// TwinCAT 3 PLC project VisionPLC
// ProgramVersion: 3.1.4024.0
// libraries:
//   Tc2_Standard, * (Beckhoff Automation GmbH)
//   Tc2_System, * (Beckhoff Automation GmbH)
//   Tc2_Utilities, * (Beckhoff Automation GmbH)
//   Tc3_Module, * (Beckhoff Automation GmbH)
//   Tc3_Vision, * (Beckhoff Automation GmbH)
// project tree:
//   DUTs/ ST_CSV_Record.TcDUT
//   GVLs/ GVL.TcGVL
//   / PlcTask.TcTTO
//   POUs/ Barcode.TcPOU, MAIN.TcPOU, P_TextModeWrite.TcPOU, QRCODE.TcPOU
// real-time tasks:
//   TASK PlcTask: cycle T#10ms, priority 20, ADS port 350
//   TASK VnTask ImgAcq (FileSource1): cycle T#10ms, priority 5, ADS port 351

CONFIGURATION VisionPLC
    RESOURCE PLC ON TwinCAT3
        TASK PlcTask(INTERVAL := T#10ms, PRIORITY := 20);
        PROGRAM MAIN WITH PlcTask : MAIN;
    END_RESOURCE
END_CONFIGURATION

// ---- DUTs/ST_CSV_Record.TcDUT
TYPE ST_CSV_Record :
STRUCT
sName 	: T_MaxString 	:= '';
	nNumber	: UDINT 		:= 0;
	fPos	: LREAL 		:= 0.0;
	bOP		: BOOL 			:= FALSE;
	sDesc	: STRING(40)	:= '';
	data	: ARRAY[0..7] OF BYTE;
END_STRUCT
END_TYPE

// ---- GVLs/GVL.TcGVL
{attribute 'qualified_only'}
VAR_GLOBAL CONSTANT
	MAX_CSV_ROWS 			: UDINT := 10;
	MAX_CSV_COLUMNS 		: UDINT := 5;
	MAX_CSV_FIELD_LENGTH	: UDINT := 100;
END_VAR

// ---- POUs/MAIN.TcPOU

PROGRAM MAIN
VAR
	//fbfilesource                                    : FB_VN_FileSourceControl;	
	CAMERA 											: FB_VN_FileSourceControl;	
	raw_image										: ITcVnImage;	
	WORKED_image										: ITcVnImage;	
	ipImageIn              						    :   ITcVnImage;
	display_raw_image								: ITcVnDisplayableImage;		
	
	ipcontours										: ITcVnContainer;	
	number_of_elements								: ULINT;	
	hr, hr1											: HRESULT;	
	cState 											: ETcVnCameraState;	
	green_color										: TcVnVector4_LREAL := [0,255,0,0];	
	Bcolor										: TcVnVector4_LREAL := [100,0,0,0];
	stext											: STRING;
	
	
//	raw_image           :    ITcVnImage;

// QR Code
ipCodeDecodedList   :    ITcVnContainer; 
ipCodeContourList   :    ITcVnContainer;
sCodeAsString       :    STRING(255);


// Output
//sText               :    STRING;

// Color
aColorRed           :    TcVnVector4_LREAL := [255, 0, 0];
pCodeDecodedList         :   ITcVnContainer; 


eBarcodeSearchDirection   :   ETcVnBarcodeSearchDirection := TCVN_BSD_ANY;
eBarcodeType              :   ETcVnBarcodeType := TCVN_BT_EAN13;
display_barcode								: ITcVnDisplayableImage;
ipImageRes: ITcVnImage;	




// Color
aColorgreen                 :   TcVnVector4_LREAL := [0, 255, 0];

//pwrite variable
bChangeSeparatorToComma	: BOOL := FALSE;
END_VAR

IF bChangeSeparatorToComma THEN
	DEFAULT_CSV_FIELD_SEP := 16#2C;(* Comma ASCII code *)
ELSE
	DEFAULT_CSV_FIELD_SEP := 16#3B;(* Semicolon ASCII code *)
END_IF




//camera code 
cState 				:= CAMERA.GetState();

CASE cState OF
	

TCVN_CS_INITIAL, TCVN_CS_OPENING, TCVN_CS_OPENED, TCVN_CS_STARTACQUISITION :

 	hr  := CAMERA.StartAcquisition();  // start Camera acquisition



TCVN_CS_ACQUIRING:
	HR := CAMERA.GetCurrentImage(raw_image);   //get image from file source 
	ipImageIn := raw_image;   //get image from file source 
	
	 IF SUCCEEDED(HR) AND ipImageIn <> 0 THEN
		 
		
// Check if the function was executed successfully 	

		

		(*hr := F_VN_ConvertColorSpace(raw_image, worked_image, TCVN_CST_RGB_TO_GRAY, hr);
		hr := F_VN_FindContours(worked_image, ipcontours, hr);
		hr := F_VN_GetNumberOfElements(ipcontours,number_of_elements, hr);
		hr := F_VN_DrawContours(ipcontours,-1,raw_image,green_color,2, hr);
		
		stext := ULINT_TO_STRING(number_of_elements);
		
		hr := F_VN_PutText(STEXT, raw_image, 70,270,TCVN_FT_HERSHEY_COMPLEX,2 , Bcolor, hr);
		
	END_IF

		hr :=  F_VN_CopyIntoDisplayableImage(raw_image, display_raw_image, hr); *)
	
 		
	//Barcode();	
 	QRCODE();
	 	END_IF

TCVN_CS_ERROR:	

	hr 	:= CAMERA.Reset();
END_CASE

END_PROGRAM

// ---- POUs/QRCODE.TcPOU
PROGRAM QRCODE
VAR
	hr              :    HRESULT;
	hr1				: HRESULT;
raw_image           :    ITcVnImage;
ipImageInDisp       :    ITcVnDisplayableImage;

ipImageResQR        :    ITcVnImage;
ipImageResDisp      :    ITcVnDisplayableImage;


// QR Code
ipCodeDecodedList   :    ITcVnContainer; 
ipCodeContourList   :    ITcVnContainer;
sCodeAsString       :    STRING(255);

// Watchdog
hrWD                :    HRESULT;
tStop               :    DINT := 20000;
tRest               :    DINT;

// Output
sText               :    STRING;

// Color
aColorRed           :    TcVnVector4_LREAL := [255, 0, 0];
aColorblue          :    TcVnVector4_LREAL := [0, 0, 255];

//string array
database1			: ARRAY[0..GVL.MAX_CSV_ROWS] OF STRING(GVL.MAX_CSV_FIELD_LENGTH);
i					: INT:=0 ;
j					: INT := 0;


	v1: STRING;
END_VAR

ipImageResQR := main.raw_image;
hr := F_VN_ReadQRCodeExp(main.raw_image, ipCodeDecodedList, ipCodeContourList, 1, TCVN_CSS_ONLY_NOT_INVERTED + TCVN_CSS_ONLY_NOT_FLIPPED, main.hr);
// Check if the function was executed successfully 
IF hr = S_OK THEN
    // Export Code into String
	hr 			:= F_VN_ExportSubContainer_String(ipCodeDecodedList, 0, sCodeAsString, 255, hr);
	P_TextModeWrite();
	

    // Write Code into Result Image
    hr := F_VN_PutTextExp(sCodeAsString,main.raw_image, 50, 50, ETcVnFontType.TCVN_FT_HERSHEY_PLAIN, 1, aColorRed,3, TCVN_LT_4_CONNECTED, FALSE, hr);

    // Draw Code Contour into Result Image
	 hr := F_VN_DrawContours(ipCodeContourList, -1, main.raw_image, aColorRed, 3, main.hr); 

    // Write HRESULT into Result Image
    sText := ('Qrcode read '); 
	hr := F_VN_PutTextExp(sText, main.raw_image, 200,240, ETcVnFontType.TCVN_FT_HERSHEY_PLAIN, 1, aColorblue,3, TCVN_LT_4_CONNECTED, FALSE, hr);
	hr :=  F_VN_CopyIntoDisplayableImage(main.raw_image, main.display_raw_image,hr);
	

	//hr1 := F_VN_PutTextExp(sText, ipImageRes, 60,240, ETcVnFontType.TCVN_FT_HERSHEY_PLAIN, 1, aColorblue,3, TCVN_LT_4_CONNECTED, FALSE, hr1);
	hr :=  F_VN_CopyIntoDisplayableImage(ipImageResQR, ipImageResDisp,hr);
ELSE
    // Write HRESULT into Result Image
    sText := CONCAT('QR cannot be read ', DINT_TO_STRING(hr)); 
    hr := F_VN_PutTextExp(sText, ipImageResQR, 70, 100, ETcVnFontType.TCVN_FT_HERSHEY_PLAIN, 1, aColorRed,3, TCVN_LT_4_CONNECTED, FALSE, hr);
	hr :=  F_VN_CopyIntoDisplayableImage(ipImageResQR, ipImageResDisp,hr);
END_IF

END_PROGRAM

// ---- POUs/P_TextModeWrite.TcPOU
(* Writing of CSV file in text mode. None of the field value is containing any non-printing control characters like line feed, carriage return, quotation marks, semicolon... *)
PROGRAM P_TextModeWrite
VAR
	bWrite			: BOOL := FALSE;(* Rising edge starts program execution *)
	sNetId			: T_AmsNetId := '';	(* TwinCAT system network address *)
	sFileName		: T_MaxString := 'C:\Users\AviNoronha\Desktop\GIT1\SAVING A CSV FILE\CSV\TextModeGen.csv';(* CSV destination file path and name *)
	sCSVLine		: T_MaxString := '';(* Single CSV text line (row, record), we are using string as record buffer (your are able to see created fields) *)
	sCSVField		: T_MaxString := '';(* Single CSV field value (column, record field) *)
	bBusy			: BOOL;
	bError			: BOOL;
	nErrId			: UDINT;
	nRow	 		: UDINT 	:= 0;(* Row number (record) *)
	nColumn			: UDINT 	:= 0;(* Column number (record field) *)
	hFile			: UINT		:= 0;(* File handle of the source file *)
	step			: DWORD 	:= 0;
	fbFileOpen		: FB_FileOpen;(* Opens file *)
	fbFileClose		: FB_FileClose;(* Closes file *)
	fbFilePuts		: FB_FilePuts;(* Writes one record (line) *)
	fbWriter		: FB_CSVMemBufferWriter;(* Helper function block used to create CSV data bytes (single record line) *)

	database		: ARRAY[0..GVL.MAX_CSV_ROWS, 0..GVL.MAX_CSV_COLUMNS ] OF STRING(GVL.MAX_CSV_FIELD_LENGTH);

    i: INT ;
	j: INT ;
	DelayCounter: INT := 0;
	DelayDuration: INT := 10000;
	v2: STRING;
END_VAR

//IF i<= 10 AND j<=5 THEN
FOR i := 0 TO 10 DO
	
    (* Loop through the columns (5) *)
    FOR j := 0 TO 5 DO
        (* Access and work with the array element *)
		v2 :=  database[i, j];
		IF v2 <> QRCODE.v1 THEN
			database[i, j] := QRCODE.sCodeAsString;  (* Example operation, replace with your logic *)
		END_IF		
    END_FOR
END_FOR
//END_IF
//database[0,1] := QRcode.sCodeAsString; 

(*IF i<= 10 AND j<=5 THEN
	database[i, j] := QRCODE.sCodeAsString;
	i := i+1;
	j := j+1;
	
END_IF*)
CASE step OF
	0:	(* Wait for rising edge at bWrite variable *)
		IF bWrite THEN
			bWrite 	:= FALSE;
			bBusy 	:= TRUE;
			bError	:= FALSE;
			nErrId	:= 0;
			hFile	:= 0;
			nRow	:= 0;
			nColumn	:= 0;
			step 	:= 1;
		END_IF

	1:	(* Open source file *)
		fbFileOpen(  bExecute := FALSE  );
		fbFileOpen( sNetId := sNetId, sPathName := sFileName, nMode := FOPEN_MODEWRITE OR FOPEN_MODETEXT,(* Open file in TEXT mode! *)
					ePath := PATH_GENERIC, bExecute := TRUE );
		step := 2;

	2:(* Wait until open not busy *)
		fbFileOpen( bExecute := FALSE, bError => bError, nErrID => nErrID, hFile => hFile );
		IF NOT fbFileOpen.bBusy THEN
			IF NOT fbFileOpen.bError THEN
				step := 3;
			ELSE(* Error: file not found? *)
				step := 100;
			END_IF
		END_IF

	3:(* Convert one PLC record to CSV format *)
		sCSVLine := '';
		fbWriter.eCmd := eEnumCmd_First;(* Write first field value *)
		IF nRow <= gvl.MAX_CSV_ROWS THEN

			FOR nColumn := 0 TO gvl.MAX_CSV_COLUMNS BY 1 DO

				sCSVField := STRING_TO_CSVFIELD( database[ nRow, nColumn ], FALSE );(* TODO: Get field value from your application *)

				(* Add new field to the record buffer *)
				fbWriter( 	pBuffer := ADR( sCSVLine ), cbBuffer := SIZEOF( sCSVLine ) - 1, putValue := sCSVField, pValue := 0, cbValue := 0,
							bCRLF := ( nColumn = gvl.MAX_CSV_COLUMNS ) );(* bCRLF == TRUE => Write CRLF after the last field value *)
				IF fbWriter.bOk THEN
					fbWriter.eCmd := eEnumCmd_Next;(* Write next field value *)
				ELSE(* Error *)
					step := 100;
					RETURN;
				END_IF

			END_FOR(* FOR nColumn := 0... *)

			(* FB_FilePuts adds allready CR (carriage return) to the written line.
			We have to replace the $R$L characters with $L character to avoid double CR. *)
			IF RIGHT( sCSVLine, 2 ) = '$R$L' THEN
				sCSVLine := REPLACE( sCSVLine, '$L', 2, LEN( sCSVLine ) - 1 );
			END_IF

			nRow := nRow + 1;(* Increment number of created records (rows) *)
			step := 4;(* Write record to the file *)

		ELSE(* All rows written => Close file *)
			step := 10;
		END_IF

	4:	(* Write single text line *)
		fbFilePuts( bExecute := FALSE );
		fbFilePuts( sNetId := sNetId, hFile := hFile, sLine := sCSVLine, bExecute := TRUE );
		step := 5;

	5:(* Wait until write not busy *)
		fbFilePuts( bExecute := FALSE, bError => bError, nErrID => nErrID );
		IF NOT fbFilePuts.bBusy THEN
			IF NOT fbFilePuts.bError THEN
				step := 3;(* Write next record *)
			ELSE(* Error *)
				step := 100;
			END_IF
		END_IF

	10:	(* Close source file *)
		fbFileClose( bExecute := FALSE );
		fbFileClose( sNetId := sNetId, hFile := hFile, bExecute := TRUE );
		step := 11;

	11:(* Wait until close not busy *)
		fbFileClose( bExecute := FALSE, bError => bError, nErrID => nErrID );
		IF ( NOT fbFileClose.bBusy ) THEN
			hFile := 0;
			step := 100;
		END_IF

	100: (* Error or ready step => cleanup *)
		IF ( hFile <> 0 ) THEN
			step := 10; (* Close the source file *)
		ELSE
			bBusy := FALSE;
			step := 0;	(* Ready *)
		END_IF

END_CASE

END_PROGRAM

// ---- POUs/Barcode.TcPOU
PROGRAM Barcode 
VAR
	hr                        :   HRESULT;


// Barcode
ipCodeDecodedList         :   ITcVnContainer; 
ipCodeContourList         :   ITcVnContainer;
sCodeAsString             :   STRING(255);
eBarcodeSearchDirection   :   ETcVnBarcodeSearchDirection := TCVN_BSD_ANY;
eBarcodeType              :   ETcVnBarcodeType := TCVN_BT_EAN13;
display_barcode								: ITcVnDisplayableImage;
ipImageRes: ITcVnImage;	

// Watchdog
hrWD                      :   HRESULT;
tStop                     :   DINT := 50000;
tRest                     :   DINT;

// Output
sText                     :   STRING;

// Color
aColorgreen                 :   TcVnVector4_LREAL := [0, 255, 0];
END_VAR

ipImageRes := main.ipImageIn   ;


 hr := F_VN_ReadBarcodeExp(main.ipImageIn, ipCodeDecodedList, ipCodeContourList,eBarcodeType, 1,eBarcodeSearchDirection , hr);
	
IF hr = S_OK THEN	
	    // Export Code into String
    hr := F_VN_ExportSubContainer_String(ipCodeDecodedList, 0, sCodeAsString, 255, hr);

    // Write Code into Result Image
    hr := F_VN_PutTextExp(sCodeAsString, main.ipImageIn, 100, 100, ETcVnFontType.TCVN_FT_HERSHEY_PLAIN, 1, aColorgreen,3, TCVN_LT_4_CONNECTED, FALSE, hr);

    // Draw Code Contour into Result Image
    hr := F_VN_DrawContours(ipCodeContourList, -1, main.ipImageIn, aColorGreen, 3, hr);
ELSE
    // Write HRESULT into Result Image
    sText := CONCAT('NOT A BARCODE ', DINT_TO_STRING(hr)); 
    hr := F_VN_PutTextExp(sText, ipImageRes, 100, 100, ETcVnFontType.TCVN_FT_HERSHEY_PLAIN, 1, aColorgreen,3, TCVN_LT_4_CONNECTED, FALSE, hr); 
END_IF
	
	//hr := F_VN_PutTextExp(sCodeAsString, main.raw_image, 60,240, ETcVnFontType.TCVN_FT_HERSHEY_PLAIN, 1, aColorblue,3, TCVN_LT_4_CONNECTED, FALSE, hr);
	hr :=  F_VN_CopyIntoDisplayableImage(ipImageRes, display_barcode,hr);

END_PROGRAM
